SYSTEM parserTest
  (* Version 1.0, 2025-07-16, dakudryashev *)
  APPLICATION parserTestApp
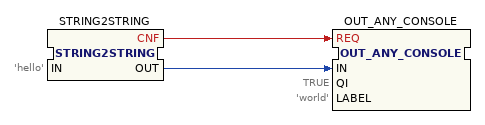
    FBS
      STRING2STRING : STRING2STRING(IN := 'hello');
      OUT_ANY_CONSOLE : OUT_ANY_CONSOLE(QI := TRUE, LABEL := 'world');
    END_FBS
    EVENT_CONNECTIONS
      STRING2STRING.CNF TO OUT_ANY_CONSOLE.REQ;
    END_CONNECTIONS
    DATA_CONNECTIONS
      STRING2STRING.OUT TO OUT_ANY_CONSOLE.IN;
    END_CONNECTIONS
  END_APPLICATION
  DEVICE FORTE_PC : FORTE_PC(MGR_ID := "localhost:61499" (* Device manager socket ID *))
    {SET_ATTRIBUTE(Profile, HOLOBLOC)}
    RESOURCE EMB_RES : EMB_RES
      EVENT_CONNECTIONS
        START.COLD TO parserTestApp.STRING2STRING.REQ;
      END_CONNECTIONS
    END_RESOURCE
  END_DEVICE
  MAPPINGS
    parserTestApp.STRING2STRING ON FORTE_PC.EMB_RES;
    parserTestApp.OUT_ANY_CONSOLE ON FORTE_PC.EMB_RES;
  END_MAPPINGS
  SEGMENTS
    Ethernet : Ethernet;
  END_SEGMENTS
  LINKS
    FORTE_PC => Ethernet;
  END_LINKS
END_SYSTEM
